(*
 	The input value will be normalize scaled from the input range [fInputMin..fInputMax] to the output range [fOutputMin..fOutputMax].	
*)
FUNCTION F_ScaleLREAL : LREAL
VAR_INPUT
	fValue 		: LREAL; //Input value
	fInputMin 	: LREAL; //Input limit Min
	fInputMax 	: LREAL; //Input limit Max
	fOutputMin 	: LREAL; //Output limit Min
	fOutputMax 	: LREAL; //Output limit Max
END_VAR

VAR
	fNormalized : LREAL;
END_VAR

VAR_OUTPUT
	bError 		: BOOL;
END_VAR

bError := (fInputMin >= fInputMax) OR (fOutputMin >= fOutputMax);

IF bError THEN
	F_ScaleLREAL := 0.0;
	RETURN;
END_IF

IF fValue < fInputMin THEN
	fNormalized := 0.0;
ELSIF fValue > fInputMax THEN
	fNormalized := 1.0;
ELSE
	fNormalized := (fValue - fInputMin) / (fInputMax - fInputMin);
END_IF

F_ScaleLREAL := fNormalized * (fOutputMax - fOutputMin) + fOutputMin;

END_FUNCTION

(* stored: Version 1.1.0.1, ProductVersion 3.1.4024.12
   POU F_ScaleLREAL: Id {846ff3a0-9af9-020d-08ce-3f919691f86f}, SpecialFunc None *)
